// TIA Portal V17 program export: 2 tag tables, 0 data types, 1 data blocks, 1 code blocks (in call order from the OBs), 0 instance data blocks

VAR_GLOBAL   // PLC tag table "Default tag table"
END_VAR

VAR_GLOBAL   // PLC tag table "Tag table_1"
END_VAR

DATA_BLOCK "Data_block_1"   // DB1
{ S7_Optimized_Access := 'TRUE' }
VERSION : 0.1
// stored: AutoNumber true, DBAccessibleFromOPCUA true, IsOnlyStoredInLoadMemory false, IsRetainMemResEnabled false, IsWriteProtectedInAS false, MemoryReserve 100
   VAR
      Tint : Int;
      Tbool : Bool;
      Treal : Real;
   END_VAR
BEGIN
END_DATA_BLOCK

ORGANIZATION_BLOCK "Main"   // OB1, LAD, ProgramCycle
TITLE = "Main Program Sweep (Cycle)"
{ S7_Optimized_Access := 'TRUE' }
VERSION : 0.1
// stored: AutoNumber true, IsIECCheckEnabled false, SetENOAutomatically false
   VAR_INPUT
      Initial_Call : Bool;   // Initial call of this OB
      Remanence : Bool;   // =True, if remanent data are available
   END_VAR
BEGIN

REGION Network 1
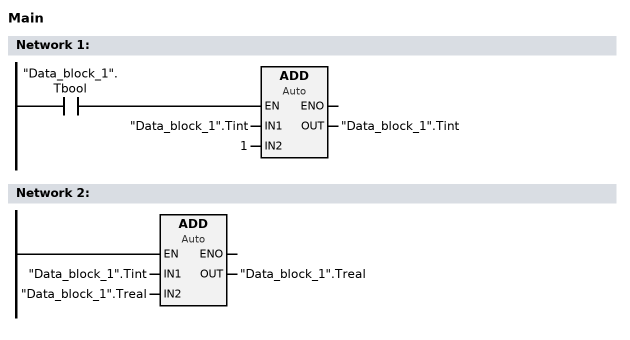
   RUNG wire#powerrail
      Contact( "Data_block_1".Tbool )
      Add(in1 := "Data_block_1".Tint, in2 := 1, out => "Data_block_1".Tint)
   END_RUNG
   // the same network as SCL:
   IF "Data_block_1".Tbool THEN "Data_block_1".Tint := "Data_block_1".Tint + 1; END_IF;
END_REGION

REGION Network 2
   RUNG wire#powerrail
      Add(in1 := "Data_block_1".Tint, in2 := "Data_block_1".Treal, out => "Data_block_1".Treal)
   END_RUNG
   // the same network as SCL:
   "Data_block_1".Treal := "Data_block_1".Tint + "Data_block_1".Treal;
END_REGION
END_ORGANIZATION_BLOCK
